FUNCTION_BLOCK FB_PDxxSimulation
VAR_INPUT
	Parameters								: ST_PDxx_SimulationParameters;
	RxPDO_1_6040h_ControlWord  				: UINT;
	RxPDO_1_6060h_ModesOfOperation  		: SINT;
	RxPDO_1_3202h_MotorDriveSubmodeSelect  	: UDINT;
	RxPDO_2_607Ah_TargetPosition  			: DINT;
	RxPDO_2_6081h_ProfileVelocity			: UDINT;
	RxPDO_3_6042h_TargetVelocity			: INT;
	RxPDO_4_60FEh_DigitalOutputs			: UDINT;

END_VAR
VAR_OUTPUT
	TxPDO_1_6041h_StatusWord  				: UINT;
	TxPDO_1_6061h_ModesOfOperationDisplay  	: SINT;
	TxPDO_2_6064h_PositionActualValue  		: DINT;
	TxPDO_3_6044h_VelocityActualValue  		: INT;
	TxPDO_4_60FDh_DigitalInputs  			: UDINT;

END_VAR
VAR
	stControlWord		: ST_PDxx_ControlWord;
	stStatusWord		: ST_PDxx_StatusWord;
	eTransition			: E_PDxx_TransitionCommand;
	trExecuteMove		: R_TRIG;
	bPositionMoveActive	: BOOL;
	nPosition			: LREAL;
	eState				: E_PDxx_State				:= E_PDxx_State.SWITCH_ON_DISABLED;
	eModesOfOperation	: E_PDxx_ModesOfOperation	:= E_PDxx_ModesOfOperation.NO_MODE_CHANGE_OR_NO_MODE_ASSIGNED;
END_VAR


A_ParseControlWord();
A_ParseTransition();
A_Motor();
A_SetStatusWord();

ACTION A_Motor:

IF eState = E_PDxx_State.OPERATION_ENABLED THEN
	CASE eModesOfOperation OF
		E_PDxx_ModesOfOperation.VELOCITY_MODE:
			VelocityMode();
		E_PDxx_ModesOfOperation.PROFILE_POSITION_MODE:
			ProfilePositionMode();
	END_CASE
ELSE
	TxPDO_3_6044h_VelocityActualValue := 0;
END_IF

TxPDO_2_6064h_PositionActualValue := LREAL_TO_DINT(nPosition);
END_ACTION

ACTION A_ParseControlWord:
 stControlWord.SwitchedOn_bit_0				:= RxPDO_1_6040h_ControlWord.0;
 stControlWord.EnableVoltage_bit_1			:= RxPDO_1_6040h_ControlWord.1;
 stControlWord.QuickStop_bit_2				:= RxPDO_1_6040h_ControlWord.2;
 stControlWord.EnableOperation_bit_3		:= RxPDO_1_6040h_ControlWord.3;
 stControlWord.OperationModeSpecific_bit_4	:= RxPDO_1_6040h_ControlWord.4;
 stControlWord.OperationModeSpecific_bit_5	:= RxPDO_1_6040h_ControlWord.5;
 stControlWord.OperationModeSpecific_bit_6	:= RxPDO_1_6040h_ControlWord.6;
 stControlWord.FaultReset_bit_7				:= RxPDO_1_6040h_ControlWord.7;
 stControlWord.Halt_bit_8					:= RxPDO_1_6040h_ControlWord.8;
 stControlWord.OperationModeSpecific_bit_9	:= RxPDO_1_6040h_ControlWord.9;
END_ACTION

ACTION A_ParseTransition:
IF
	stControlWord.FaultReset_bit_7 = TRUE AND
   	eTransition <> E_PDxx_TransitionCommand.FAULT_RESET THEN
		eTransition := E_PDxx_TransitionCommand.FAULT_RESET;
ELSIF
	stControlWord.SwitchedOn_bit_0 = FALSE AND
	stControlWord.EnableVoltage_bit_1 = TRUE AND
	stControlWord.QuickStop_bit_2 = TRUE AND
	stControlWord.FaultReset_bit_7 = FALSE THEN
		eTransition := E_PDxx_TransitionCommand.SHUTDOWN;
ELSIF
	stControlWord.SwitchedOn_bit_0 = TRUE AND
	stControlWord.EnableVoltage_bit_1 = TRUE AND
	stControlWord.QuickStop_bit_2 = TRUE AND
	stControlWord.EnableOperation_bit_3 = FALSE AND
	stControlWord.FaultReset_bit_7 = FALSE THEN
		eTransition := E_PDxx_TransitionCommand.SWITCH_ON;
ELSIF
	stControlWord.EnableVoltage_bit_1 = FALSE AND
	stControlWord.FaultReset_bit_7 = FALSE THEN
		eTransition := E_PDxx_TransitionCommand.DISABLE_VOLTAGE;
ELSIF
	stControlWord.EnableVoltage_bit_1 = TRUE AND
	stControlWord.QuickStop_bit_2 = FALSE AND
	stControlWord.FaultReset_bit_7 = FALSE THEN
		eTransition := E_PDxx_TransitionCommand.QUICK_STOP;
ELSIF
	stControlWord.SwitchedOn_bit_0 = TRUE AND
	stControlWord.EnableVoltage_bit_1 = TRUE AND
	stControlWord.QuickStop_bit_2 = TRUE AND
	stControlWord.EnableOperation_bit_3 = TRUE AND
	stControlWord.FaultReset_bit_7 = FALSE THEN
		eTransition := E_PDxx_TransitionCommand.ENABLE_OPERATION;
END_IF

CASE eTransition OF
	E_PDxx_TransitionCommand.FAULT_RESET:
		IF eState = E_PDxx_State.FAULT THEN
			eState := E_PDxx_State.SWITCH_ON_DISABLED;
		END_IF
	E_PDxx_TransitionCommand.SHUTDOWN:
		IF eState = E_PDxx_State.SWITCH_ON_DISABLED OR
		   eState = E_PDxx_State.SWITCHED_ON OR
		   eState = E_PDxx_State.OPERATION_ENABLED THEN
			eState := E_PDxx_State.READY_TO_SWITCH_ON;
		END_IF
	E_PDxx_TransitionCommand.SWITCH_ON:
		IF eState = E_PDxx_State.READY_TO_SWITCH_ON OR
		   eState = E_PDxx_State.OPERATION_ENABLED THEN
			eState := E_PDxx_State.SWITCHED_ON;
		END_IF
	E_PDxx_TransitionCommand.DISABLE_VOLTAGE:
		IF eState = E_PDxx_State.READY_TO_SWITCH_ON OR
		   eState = E_PDxx_State.SWITCHED_ON OR
		   eState = E_PDxx_State.OPERATION_ENABLED OR
		   eState = E_PDxx_State.QUICK_STOP_ACTIVE THEN
			eState := E_PDxx_State.SWITCH_ON_DISABLED;
		END_IF
	E_PDxx_TransitionCommand.QUICK_STOP:
		IF eState = E_PDxx_State.OPERATION_ENABLED THEN
			eState := E_PDxx_State.QUICK_STOP_ACTIVE;
		END_IF
	E_PDxx_TransitionCommand.ENABLE_OPERATION:
		IF eState = E_PDxx_State.SWITCHED_ON THEN
			eState := E_PDxx_State.OPERATION_ENABLED;
		END_IF
END_CASE

IF eState = E_PDxx_State.SWITCH_ON_DISABLED OR
   eState = E_PDxx_State.READY_TO_SWITCH_ON OR
   eState = E_PDxx_State.SWITCHED_ON THEN
   	TxPDO_1_6061h_ModesOfOperationDisplay := RxPDO_1_6060h_ModesOfOperation;
END_IF

CASE TxPDO_1_6061h_ModesOfOperationDisplay OF
	-2: eModesOfOperation := E_PDxx_ModesOfOperation.AUTO_SETUP;
	-1: eModesOfOperation := E_PDxx_ModesOfOperation.CLOCK_DIRECTION_MODE;
	0: eModesOfOperation := E_PDxx_ModesOfOperation.NO_MODE_CHANGE_OR_NO_MODE_ASSIGNED;
	1: eModesOfOperation := E_PDxx_ModesOfOperation.PROFILE_POSITION_MODE;
	2: eModesOfOperation := E_PDxx_ModesOfOperation.VELOCITY_MODE;
	3: eModesOfOperation := E_PDxx_ModesOfOperation.PROFILE_VELOCITY_MODE;
	4: eModesOfOperation := E_PDxx_ModesOfOperation.PROFILE_TORQUE_MODE;
	5: eModesOfOperation := E_PDxx_ModesOfOperation.RESERVED;
	6: eModesOfOperation := E_PDxx_ModesOfOperation.HOMING_MODE;
	7: eModesOfOperation := E_PDxx_ModesOfOperation.INTERPOLATED_POSITION_MODE;
	8: eModesOfOperation := E_PDxx_ModesOfOperation.CYCLIC_SYNCHRONOUS_POSITION_MODE;
	9: eModesOfOperation := E_PDxx_ModesOfOperation.CYCLIC_SYNCHRONOUS_VELOCITY_MODE;
	10: eModesOfOperation := E_PDxx_ModesOfOperation.CYCLIC_SYNCHRONOUS_TORQUE_MODE;	
END_CASE
END_ACTION

ACTION A_SetStatusWord:
CASE eState OF
	E_PDxx_State.NOT_READY_TO_SWITCH_ON:
		stStatusWord.ReadyToSwitchOn	:= FALSE;
		stStatusWord.SwitchedOn			:= FALSE;
		stStatusWord.OperationEnabled	:= FALSE;
		stStatusWord.Fault				:= FALSE;
//		stStatusWord.VoltageEnabled		:= FALSE;
//		stStatusWord.QuickStop			:= FALSE;
		stStatusWord.SwitchOnDisabled	:= FALSE;
	E_PDxx_State.SWITCH_ON_DISABLED:
		stStatusWord.ReadyToSwitchOn	:= FALSE;
		stStatusWord.SwitchedOn			:= FALSE;
		stStatusWord.OperationEnabled	:= FALSE;
		stStatusWord.Fault				:= FALSE;
//		stStatusWord.VoltageEnabled		:= FALSE;
//		stStatusWord.QuickStop			:= FALSE;
		stStatusWord.SwitchOnDisabled	:= TRUE;
	E_PDxx_State.READY_TO_SWITCH_ON:
		stStatusWord.ReadyToSwitchOn	:= TRUE;
		stStatusWord.SwitchedOn			:= FALSE;
		stStatusWord.OperationEnabled	:= FALSE;
		stStatusWord.Fault				:= FALSE;
//		stStatusWord.VoltageEnabled		:= FALSE;
		stStatusWord.QuickStop			:= TRUE;
		stStatusWord.SwitchOnDisabled	:= FALSE;
	E_PDxx_State.SWITCHED_ON:
		stStatusWord.ReadyToSwitchOn	:= TRUE;
		stStatusWord.SwitchedOn			:= TRUE;
		stStatusWord.OperationEnabled	:= FALSE;
		stStatusWord.Fault				:= FALSE;
//		stStatusWord.VoltageEnabled		:= FALSE;
		stStatusWord.QuickStop			:= TRUE;
		stStatusWord.SwitchOnDisabled	:= FALSE;
	E_PDxx_State.OPERATION_ENABLED:
		stStatusWord.ReadyToSwitchOn	:= TRUE;
		stStatusWord.SwitchedOn			:= TRUE;
		stStatusWord.OperationEnabled	:= TRUE;
		stStatusWord.Fault				:= FALSE;
//		stStatusWord.VoltageEnabled		:= FALSE;
		stStatusWord.QuickStop			:= TRUE;
		stStatusWord.SwitchOnDisabled	:= FALSE;
	E_PDxx_State.QUICK_STOP_ACTIVE:
		stStatusWord.ReadyToSwitchOn	:= TRUE;
		stStatusWord.SwitchedOn			:= TRUE;
		stStatusWord.OperationEnabled	:= TRUE;
		stStatusWord.Fault				:= FALSE;
//		stStatusWord.VoltageEnabled		:= FALSE;
		stStatusWord.QuickStop			:= FALSE;
		stStatusWord.SwitchOnDisabled	:= FALSE;
	E_PDxx_State.FAULT_REACTION_ACTIVE:
		stStatusWord.ReadyToSwitchOn	:= TRUE;
		stStatusWord.SwitchedOn			:= TRUE;
		stStatusWord.OperationEnabled	:= TRUE;
		stStatusWord.Fault				:= TRUE;
//		stStatusWord.VoltageEnabled		:= FALSE;
//		stStatusWord.QuickStop			:= FALSE;
		stStatusWord.SwitchOnDisabled	:= FALSE;
	E_PDxx_State.FAULT:
		stStatusWord.ReadyToSwitchOn	:= FALSE;
		stStatusWord.SwitchedOn			:= FALSE;
		stStatusWord.OperationEnabled	:= FALSE;
		stStatusWord.Fault				:= TRUE;
//		stStatusWord.VoltageEnabled		:= FALSE;
//		stStatusWord.QuickStop			:= FALSE;
		stStatusWord.SwitchOnDisabled	:= FALSE;
END_CASE

// Set more statusword bits if necessary for simulation, for example target reached and closed loop???

TxPDO_1_6041h_StatusWord.0 := stStatusWord.ReadyToSwitchOn;
TxPDO_1_6041h_StatusWord.1 := stStatusWord.SwitchedOn;
TxPDO_1_6041h_StatusWord.2 := stStatusWord.OperationEnabled;
TxPDO_1_6041h_StatusWord.3 := stStatusWord.Fault;
TxPDO_1_6041h_StatusWord.4 := stStatusWord.VoltageEnabled;
TxPDO_1_6041h_StatusWord.5 := stStatusWord.QuickStop;
TxPDO_1_6041h_StatusWord.6 := stStatusWord.SwitchOnDisabled;
TxPDO_1_6041h_StatusWord.7 := stStatusWord.Warning;
TxPDO_1_6041h_StatusWord.8 := stStatusWord.Synchronization;
TxPDO_1_6041h_StatusWord.9 := stStatusWord.Remote;
TxPDO_1_6041h_StatusWord.10 := stStatusWord.TargetReached;
TxPDO_1_6041h_StatusWord.11 := stStatusWord.InternalLimitReached;
TxPDO_1_6041h_StatusWord.12 := stStatusWord.OperationModeSpecific_bit12;
TxPDO_1_6041h_StatusWord.13 := stStatusWord.OperationModeSpecific_bit13;
TxPDO_1_6041h_StatusWord.15 := stStatusWord.ClosedLoopAvailable;
END_ACTION

METHOD PRIVATE ProfilePositionMode
VAR
	nDeltaPosition : LREAL;
	nTargetPosition : LREAL;
END_VAR
trExecuteMove.CLK := stControlWord.OperationModeSpecific_bit_4;
IF trExecuteMove.Q = TRUE THEN
	bPositionMoveActive := TRUE;
	stStatusWord.OperationModeSpecific_bit12 := TRUE;
END_IF

IF bPositionMoveActive = TRUE THEN
	IF RxPDO_2_6081h_ProfileVelocity < 0 THEN
		TxPDO_3_6044h_VelocityActualValue  := -UDINT_TO_INT(RxPDO_2_6081h_ProfileVelocity);
	ELSE
		TxPDO_3_6044h_VelocityActualValue  :=  UDINT_TO_INT(RxPDO_2_6081h_ProfileVelocity);
	END_IF
	
	nTargetPosition := DINT_TO_LREAL(RxPDO_2_607Ah_TargetPosition);
	nDeltaPosition := nPosition + INT_TO_LREAL(TxPDO_3_6044h_VelocityActualValue) * Parameters.nMMPerSecondPerVelUnit * Parameters.nSecondsPerSimStep;

	IF nPosition < nTargetPosition AND
	   nPosition + nDeltaPosition >=  nTargetPosition THEN
		nPosition := nTargetPosition;
		stStatusWord.TargetReached := TRUE;
		bPositionMoveActive := FALSE;
		RETURN;
	END_IF
	
	IF nPosition > nTargetPosition AND
	   nPosition + nDeltaPosition <=  nTargetPosition THEN
		nPosition := nTargetPosition;
		stStatusWord.TargetReached := TRUE;
		bPositionMoveActive := FALSE;
		RETURN;
	END_IF
	
	nPosition := nPosition + nDeltaPosition; 
	
	IF nPosition < Parameters.nPositionMin THEN
		nPosition := Parameters.nPositionMin;
		TxPDO_3_6044h_VelocityActualValue := 0;
	END_IF
	
	IF nPosition > Parameters.nPositionMax THEN
		nPosition := Parameters.nPositionMax;
		TxPDO_3_6044h_VelocityActualValue := 0;
	END_IF

END_IF

IF stControlWord.OperationModeSpecific_bit_4 = FALSE THEN
	stStatusWord.OperationModeSpecific_bit12 := FALSE;
END_IF
END_METHOD


METHOD PRIVATE VelocityMode

TxPDO_3_6044h_VelocityActualValue  :=  RxPDO_3_6042h_TargetVelocity;

nPosition := nPosition + DINT_TO_LREAL(TxPDO_3_6044h_VelocityActualValue) * Parameters.nMMPerSecondPerVelUnit * Parameters.nSecondsPerSimStep; 

IF nPosition < Parameters.nPositionMin THEN
	nPosition := Parameters.nPositionMin;
	TxPDO_3_6044h_VelocityActualValue := 0;
END_IF

IF nPosition > Parameters.nPositionMax THEN
	nPosition := Parameters.nPositionMax;
	TxPDO_3_6044h_VelocityActualValue := 0;
END_IF
END_METHOD

END_FUNCTION_BLOCK

(* stored: Version 1.1.0.1, ProductVersion 3.1.4024.12
   POU FB_PDxxSimulation: Id {a4499cb8-8c92-424d-9fa9-d12ea02e01ac}, SpecialFunc None
   Action A_Motor: Id {4d1f7ea6-bdce-4b54-a84e-dc840b18b146}
   Action A_ParseControlWord: Id {229f2ec5-6b2f-408c-ac5a-f4889636f2ac}
   Action A_ParseTransition: Id {0645cff6-4128-4ef8-9dc4-ced99a62c158}
   Action A_SetStatusWord: Id {86854303-5eba-44b9-84b6-5cf55c4c8c77}
   Method ProfilePositionMode: Id {a50ad241-0646-49e3-ace3-5d2da85d4833}
   Method VelocityMode: Id {9037df63-8ba2-4360-b635-c99c1b1ed146} *)
